// TIA Portal V16 export
// export: Created 2024-12-03T15:41:41.1683802Z, ExportSetting WithDefaults, DisplayName Totally Integrated Automation Portal, DisplayVersion V16 Update 6, DisplayName TIA Portal Version Control Interface, DisplayVersion V16 Update 2, DisplayName TIA Portal Openness, DisplayVersion V16 Update 6, DisplayName TIA Portal Teamcenter Gateway, DisplayVersion V16, DisplayName SINAMICS Startdrive Advanced, DisplayVersion V16 Update 5, DisplayName SINAMICS Startdrive G130, G150, S120, S150, SINAMICS MV, S210, DisplayVersion V16 Update 5, DisplayName SINAMICS Startdrive G110M, G120, G120C, G120D, G120P, G115D, DisplayVersion V16 Update 5, DisplayName STEP 7 Professional, DisplayVersion V16 Update 6, DisplayName STEP 7 Safety, DisplayVersion V16, DisplayName WinCC Advanced / Unified PC, DisplayVersion V16 Update 6
FUNCTION_BLOCK "HeartBeatButton_FB"   // FB24, SCL
{ S7_Optimized_Access := 'TRUE' }
VERSION : 0.1
// stored: AutoNumber true, IsIECCheckEnabled false, IsRetainMemResEnabled false, MemoryReserve 100, SetENOAutomatically false, UDAEnableTagReadback false
   VAR_INPUT
      I_BeatSpeed : Time := t#1s;
   END_VAR
   VAR_IN_OUT
      IO_Beat : "HeartBeatButton_UDT";
   END_VAR
   VAR
      beater : TON_TIME;
      prevValue { S7_SetPoint := 'True'} : Byte;
   END_VAR
BEGIN
   #beater(IN := #IO_Beat.beat > 0 AND #prevValue = #IO_Beat.beat,
           PT := #I_BeatSpeed);

   IF #beater.Q THEN
       #IO_Beat.beat := 0;
   END_IF;

   IF #IO_Beat.beat > 0 THEN
       #IO_Beat.state := 1;
   END_IF;

   IF #IO_Beat.beat = 0 THEN
       #IO_Beat.state := 0;
   END_IF;

   #prevValue := #IO_Beat.beat;
END_FUNCTION_BLOCK
